PROGRAM MAIN
VAR
END_VAR

END_PROGRAM

(* stored: Version 1.1.0.1
   POU MAIN: Id {88103d41-d565-4349-8789-4d54234d4e5a} *)
